// TIA Portal V19 export
TYPE "LEXCHANGETRAY_typeScanner_cmd"
// stored: Access Published
   STRUCT
      simActive : Bool;
      reset : Bool;
      cmdStep : Int;
   END_STRUCT;
END_TYPE
